// TwinCAT 3 PLC project RFID
// ProgramVersion: 3.1.4024.0
// libraries:
//   Tc2_Standard, * (Beckhoff Automation GmbH)
//   Tc2_System, * (Beckhoff Automation GmbH)
//   Tc2_TcpIp, * (Beckhoff Automation GmbH)
//   Tc2_Utilities, * (Beckhoff Automation GmbH)
//   Tc3_Module, * (Beckhoff Automation GmbH)
// project tree:
//   / PlcTask.TcTTO
//   POUs/ FB_RRU7001.TcPOU, FB_TcpClient.TcPOU, I_TcpClient.TcIO, MAIN.TcPOU
// real-time tasks:
//   TASK PlcTask: cycle T#10ms, priority 20, ADS port 350

CONFIGURATION RFID
    RESOURCE PLC ON TwinCAT3
        TASK PlcTask(INTERVAL := T#10ms, PRIORITY := 20);
        PROGRAM MAIN WITH PlcTask : MAIN;
    END_RESOURCE
END_CONFIGURATION

// ---- POUs/I_TcpClient.TcIO
INTERFACE I_TcpClient

METHOD M_Connect
VAR_INPUT
	sIP   : STRING;
    nPort : UINT;
END_VAR
END_METHOD

METHOD M_Cyclic
VAR_INPUT
END_VAR
END_METHOD

METHOD M_GetData : UDINT;
VAR_INPUT
	pDest : POINTER TO BYTE;
    nSize : UDINT;
END_VAR
END_METHOD

PROPERTY P_HasNewData : bool
GET
END_GET
END_PROPERTY

END_INTERFACE

// ---- POUs/MAIN.TcPOU
PROGRAM MAIN
VAR
	fbReader : FB_RRU7001;
END_VAR

fbReader();

END_PROGRAM

// ---- POUs/FB_RRU7001.TcPOU
FUNCTION_BLOCK FB_RRU7001
VAR
    fbNetwork       : FB_TcpClient;
    arrRawData      : ARRAY[0..255] OF BYTE;
    nRecBytes       : UDINT;
    
    bInit           : BOOL := TRUE;
    i               : INT;
    sUID            : STRING(100); 
END_VAR

IF bInit THEN
    fbNetwork.M_Connect(sIP := '192.168.1.190', nPort := 6000); 
    bInit := FALSE;
END_IF

fbNetwork.M_Cyclic();

IF fbNetwork.P_HasNewData THEN
    nRecBytes := fbNetwork.M_GetData(pDest := ADR(arrRawData), nSize := SIZEOF(arrRawData));

    IF nRecBytes > 0 THEN
        sUID := '';
        FOR i := 6 TO 17 DO
            sUID := CONCAT(sUID, BYTE_TO_HEXSTR(in := arrRawData[i], iPrecision := 2, bLoCase := FALSE));
            IF i < 17 THEN 
                sUID := CONCAT(sUID, ' '); 
            END_IF
        END_FOR
    END_IF
END_IF

END_FUNCTION_BLOCK

// ---- POUs/FB_TcpClient.TcPOU
FUNCTION_BLOCK FB_TcpClient IMPLEMENTS I_TcpClient
VAR_INPUT
END_VAR
VAR_OUTPUT
END_VAR
VAR
	fbConnect    : FB_SocketConnect;
    fbReceive    : FB_SocketReceive;
    hSocket      : T_HSOCKET;
    
    nState       : INT;
    bCmdConnect  : BOOL;
	sTargetIP	  : STRING;
	nTargetPort	: UINT;
    
    arrBuffer    : ARRAY[0..255] OF BYTE;
    nRxBytes     : UDINT;
    bDataReady   : BOOL;
END_VAR

{warning 'add method implementation '}
METHOD M_Connect
VAR_INPUT
	sIP	    : STRING;
	nPort	: UINT;
END_VAR
sTargetIP := sIP;
nTargetPort := nPort;
bCmdConnect := TRUE;
END_METHOD

{warning 'add method implementation '}
METHOD M_Cyclic
CASE nState OF
    0: 
        IF bCmdConnect THEN
            bCmdConnect := FALSE;
            nState := 10;
        END_IF
        
    10: 
        fbConnect(sSrvNetId := '', sRemoteHost := sTargetIP, nRemotePort := nTargetPort, bExecute := TRUE, tTimeout := T#3S);
        IF NOT fbConnect.bBusy THEN
            IF NOT fbConnect.bError THEN
                hSocket := fbConnect.hSocket;
                nState := 20; 
            ELSE
                nState := 99; 
            END_IF
            fbConnect(bExecute := FALSE);
        END_IF
          
    20: 
        IF NOT fbReceive.bBusy THEN
            fbReceive.bExecute := TRUE;
        END_IF
        
        fbReceive(sSrvNetId := '', hSocket := hSocket, cbLen := SIZEOF(arrBuffer), pDest := ADR(arrBuffer), tTimeout := T#1S);
        
        IF NOT fbReceive.bBusy AND fbReceive.bExecute THEN
            IF NOT fbReceive.bError AND fbReceive.nRecBytes > 0 THEN
                nRxBytes := fbReceive.nRecBytes;
                bDataReady := TRUE; 
            END_IF
            fbReceive.bExecute := FALSE; 
            fbReceive(); 
        END_IF
END_CASE
END_METHOD

{warning 'add method implementation '}
METHOD M_GetData : UDINT;
VAR_INPUT
	pDest	: POINTER TO BYTE;
	nSize	: UDINT;
END_VAR
IF bDataReady THEN
    MEMCPY(destAddr := pDest, srcAddr := ADR(arrBuffer), n := MIN(nSize, nRxBytes));
    M_GetData  := nRxBytes;
    bDataReady := FALSE;
ELSE
    M_GetData := 0;
END_IF
END_METHOD

{warning 'add property implementation'}
PROPERTY P_HasNewData : BOOL
GET
P_HasNewData := bDataReady;
END_GET
END_PROPERTY

END_FUNCTION_BLOCK
